// TIA Portal V16 export
// export: Created 2021-11-12T13:32:40.5420966Z, ExportSetting WithDefaults, DisplayName Totally Integrated Automation Portal, DisplayVersion V16 Update 3, DisplayName TIA Portal Version Control Interface, DisplayVersion V16 Update 2, DisplayName TIA Portal Openness, DisplayVersion V16 Update 3, DisplayName SINAMICS Startdrive Advanced, DisplayVersion V16 Update 5, DisplayName SINAMICS Startdrive G130, G150, S120, S150, SINAMICS MV, S210, DisplayVersion V16 Update 5, DisplayName SINAMICS Startdrive G110M, G120, G120C, G120D, G120P, G115D, DisplayVersion V16 Update 5, DisplayName STEP 7 Professional, DisplayVersion V16 Update 3, DisplayName STEP 7 Safety, DisplayVersion V16, DisplayName WinCC UA Professional, DisplayVersion V16 Update 3
DATA_BLOCK "IDB_Station2R2"   // DB38
{ DB_Accessible_From_OPC_UA := 'FALSE' }
VERSION : 0.1
// stored: AutoNumber true, DBAccessibleFromOPCUA false, InstanceOfName Station2R2, InstanceOfType FB
"Station2R2"
   // VAR
   //    SF_RO01_Timeout : "STD_DI_Mon";
   //    SF_RO01_LubStartErr { S7_SetPoint := 'True'} : "STD_DI_Mon";
   //    "SF_CM01-BL01_Wrn" { S7_SetPoint := 'True'} : "STD_DI_Mon";
   //    "SF_CM01-BL01_Err" { S7_SetPoint := 'True'} : "STD_DI_Mon";
   //    SF_RO01 { S7_SetPoint := 'True'} : "STD_RobotABB";
   //    SF_RC01 : "STD_DriveRobotABB";
   //    SS_Edge { S7_SetPoint := 'True'} : Array[0..16] of Bool;
   //    SB1ReqServPos { ExternalAccessible := 'False'; ExternalVisible := 'False'; ExternalWritable := 'False'} : Bool;
   //    SB1ReqToolchange : Bool;
   //    SB1ReqFlush : Bool;
   //    SB1ReqFlushAux { ExternalAccessible := 'False'; ExternalVisible := 'False'; ExternalWritable := 'False'} : Bool;
   //    SB1ReqSprayMan : Bool;
   //    SB1ReqSprayManAux { ExternalAccessible := 'False'; ExternalVisible := 'False'; ExternalWritable := 'False'} : Bool;
   //    SB1CycleAutostop : Bool;
   //    SB1RobotInitialized : Bool;
   // END_VAR
BEGIN
END_DATA_BLOCK
